TYPE "UDT_ZC_RECETA_CIP_ACIDO_LIMP"
VERSION : 0.1
   STRUCT
      TiempoEmpujeADestino : Int;   // ACIDO LIMP. Tiempo de empuje a destino
      TiempoMaxVaciadoDestino : Int;   // ACIDO LIMP. Tiempo Max vaciado destino
      TiempoEmpujeDestinoACCIP : Int;   // ACIDO LIMP. Tiempoi empuje desde equipo a CIP
      TiempoLimpieza : Int;   // ACIDO LIMP. Tiempo Limpieza
      ReservaInt_1 : Int;   // ACIDO LIMP.
      ReservaInt_2 : Int;   // ACIDO LIMP.
      TemperaturaLimpieza : Real;   // ACIDO LIMP. Temperatura limpieza
      TemperaturaHisteresis : Real;   // ACIDO LIMP. Temperatura limpieza histeresis
      ConductividadDrenaje : Real;   // ACIDO LIMP. Conductividad para Drenaje
      ConductividadLimpiezaOk : Real;   // ACIDO LIMP. Conductividad limpieza Ok
      TemperaturaLimpiezaOk : Real;   // ACIDO LIMP. Temperatura limpieza Ok
   END_STRUCT;

END_TYPE

